// TwinCAT 3 PLC project washer
// ProgramVersion: 3.1.4024.0
// libraries:
//   Tc2_Standard, * (Beckhoff Automation GmbH)
//   Tc2_System, * (Beckhoff Automation GmbH)
//   Tc3_Module, * (Beckhoff Automation GmbH)
// project tree:
//   / PlcTask.TcTTO
//   POUs/ MAIN.TcPOU, POU.TcPOU
// real-time tasks:
//   TASK PlcTask: cycle T#10ms, priority 20, ADS port 350

CONFIGURATION washer
    RESOURCE PLC ON TwinCAT3
        TASK PlcTask(INTERVAL := T#10ms, PRIORITY := 20);
        PROGRAM MAIN WITH PlcTask : MAIN;
    END_RESOURCE
END_CONFIGURATION

// ---- POUs/MAIN.TcPOU
PROGRAM MAIN
VAR
END_VAR

POU();

END_PROGRAM

// ---- POUs/POU.TcPOU
PROGRAM POU
VAR
	xStart: BOOL;
	xStop: BOOL;
	xCarPresent: BOOL;	
	xOut1: BOOL;	
	xWetting: BOOL;
	xSoaping: BOOL;
	xScrubbing: BOOL;
	xRinsing: BOOL;
	xDrying: BOOL;
	WettingPhase: TP;
	SoapingPhase: TP;
	ScrubbingPhase: TP;
	RinsingPhase: TP;
	DryingPhase: TP;
END_VAR

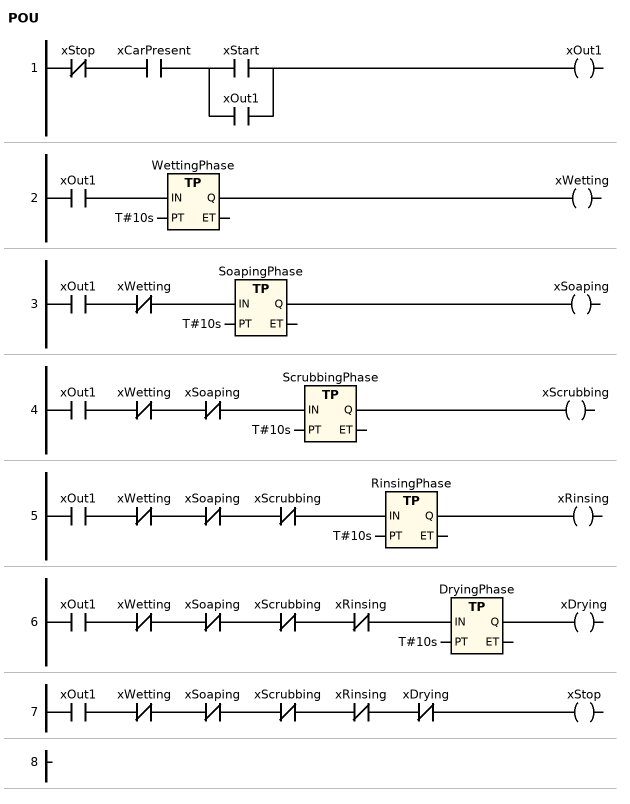
// NETWORK 1
xOut1 := NOT xStop AND xCarPresent AND (xStart OR xOut1);

// NETWORK 2
WettingPhase(IN := xOut1, PT := T#10s); // TP
xWetting := WettingPhase.Q;

// NETWORK 3
SoapingPhase(IN := xOut1 AND NOT xWetting, PT := T#10s); // TP
xSoaping := SoapingPhase.Q;

// NETWORK 4
ScrubbingPhase(IN := xOut1 AND NOT xWetting AND NOT xSoaping, PT := T#10s); // TP
xScrubbing := ScrubbingPhase.Q;

// NETWORK 5
RinsingPhase(IN := xOut1 AND NOT xWetting AND NOT xSoaping AND NOT xScrubbing, PT := T#10s); // TP
xRinsing := RinsingPhase.Q;

// NETWORK 6
DryingPhase(IN := xOut1 AND NOT xWetting AND NOT xSoaping AND NOT xScrubbing AND NOT xRinsing, PT := T#10s); // TP
xDrying := DryingPhase.Q;

// NETWORK 7
xStop := xOut1 AND NOT xWetting AND NOT xSoaping AND NOT xScrubbing AND NOT xRinsing AND NOT xDrying;

// NETWORK 8

END_PROGRAM
